// TIA Portal V17 export
// export: Created 2023-12-22T15:03:17.6906405Z, ExportSetting WithDefaults, DisplayName Totally Integrated Automation Portal, DisplayVersion V17, DisplayName TIA Portal Openness, DisplayVersion V17, DisplayName TIA Portal Version Control Interface, DisplayVersion V17, DisplayName STEP 7 Professional, DisplayVersion V17, DisplayName STEP 7 Safety, DisplayVersion V17, DisplayName WinCC Advanced, DisplayVersion V17
DATA_BLOCK "KP_REQ"   // DB6
{ S7_Optimized_Access := 'FALSE' }
VERSION : 0.1
// stored: AutoNumber true, DBAccessibleFromOPCUA true, DBAccessibleFromWebserver true, IsOnlyStoredInLoadMemory false, IsWriteProtectedInAS false
   VAR
      KP_2_1 : Array[0..15] of Bool;
      KP_2_2 : Array[0..15] of Bool;
      KP_2_3 : Array[0..15] of Bool;
      KP_2_4 : Array[0..15] of Bool;
      KP_2_5 : Array[0..15] of Bool;
      KP_2_6 : Array[0..15] of Bool;
      KP_2_7 : Array[0..15] of Bool;
      KP_2_8 : Array[0..15] of Bool;
      KP_2_9 : Array[0..15] of Bool;
      KP_2_10 : Array[0..15] of Bool;
   END_VAR
BEGIN
END_DATA_BLOCK
